Staubli VAL3: onF1Event.pgx

program onF1Event()
  local num i
  local string l_sItem
  local string l_sPage
begin
  // look if the bButton is enable
  if bButton[0]
    //
    // load Select Program
    l_sPage="Disk://instruction/PROG/page_program"
    l_sItem=""
    call loadPage(l_sPage,l_sItem)
    //
    logMsg("[KERNEL] INTERFACE:PAGE Home Page")
  endIf
end
